// TwinCAT 3 PLC project CX9240
// ProgramVersion: 3.1.4026.20
// libraries:
//   Tc2_Standard, * (Beckhoff Automation GmbH)
//   Tc2_System, * (Beckhoff Automation GmbH)
// project tree:
//   DUTs/ ST_LED.TcDUT, ST_Switch.TcDUT, U_LED.TcDUT, U_Switch.TcDUT
//   GVLs/ GVL.TcGVL
//   / PlcTask.TcTTO
//   POUs/ MAIN.TcPOU
// real-time tasks:
//   TASK PlcTask: cycle T#10ms, priority 20, ADS port 350
//   TASK Ethernet/IP Task: cycle T#1ms, priority 2, ADS port 301
// I/O:
//   DEVICE デバイス 1 (CCAT EIP Adapter(Slave)), AmsNetId 192.168.15.13.3.1
//     Box 1 (TC EtherNet/IP Slave)
//   DEVICE デバイス 3 (EtherCAT), AmsNetId 192.168.15.13.5.1
//     ターミナル 1 (EK1200) [EK1200-5000 EtherCAT Power supply (2A E-Bus)]
//       ターミナル 3 (EL6224) [EL6224 (IO Link Master)]
//       ターミナル 4 (EK1110) [EK1110 EtherCAT extension]
//     ターミナル 5 (EK1828) [EK1828 EtherCAT IO-Coupler  (1A E-Bus, 4 Ch. Dig. In, 3ms, 8 Ch. Dig. Out 24V, 0,5A)]
//       ターミナル 6 (EL3318) [EL3318 8Ch. Ana Input Thermocouple (TC)]
//       ターミナル 6 (EL9011)
// variable links:
//   (this object) <-> Device 1 (CCAT EIP Adapter(Slave))/Box 1 (TC EtherNet/IP Slave)
//     PlcTask Inputs/GVL.uLED/uiUINT <-> Assembly 1 (Input/Output)/Inputs/uiUINT
//     PlcTask Outputs/GVL.uSwitch/uiUINT <-> Assembly 1 (Input/Output)/Outputs/uiUINT

CONFIGURATION CX9240
    RESOURCE PLC ON TwinCAT3
        TASK PlcTask(INTERVAL := T#10ms, PRIORITY := 20);
        PROGRAM MAIN WITH PlcTask : MAIN;
    END_RESOURCE
END_CONFIGURATION

// ---- DUTs/ST_LED.TcDUT
TYPE ST_LED :
STRUCT
	bGreenLED		:BIT;
	bYellowLED		:BIT;
	bRedLED			:BIT;
	bWhiteLED		:BIT;
	bBlueLED		:BIT;
END_STRUCT
END_TYPE

// ---- DUTs/ST_Switch.TcDUT
TYPE ST_Switch :
STRUCT
	bGreenSwitch		:BIT;
	bYellowSwitch		:BIT;
	bRedSwitch			:BIT;
	bWhiteSwitch		:BIT;
	bBlueSwitch			:BIT;
END_STRUCT
END_TYPE

// ---- DUTs/U_LED.TcDUT
TYPE U_LED :
UNION
	uiUINT		:UINT;
	stLED		:ST_LED;
	
END_UNION
END_TYPE

// ---- DUTs/U_Switch.TcDUT
TYPE U_Switch :
UNION
	uiUINT		:UINT;
	stSwitch	:ST_Switch;
	
END_UNION
END_TYPE

// ---- GVLs/GVL.TcGVL
{attribute 'qualified_only'}
VAR_GLOBAL
	
///---Modbus TCP---
    mb_Input_Coils					:ARRAY [0..255] OF BOOL;
    mb_Output_Coils					:ARRAY [0..255] OF BOOL;
    mb_Input_Registers				:ARRAY [0..255] OF WORD;
    mb_Output_Registers				:ARRAY [0..255] OF WORD;

//---EtherNet/IP---
	uLED					AT %I*	:U_LED;
	uSwitch					AT %Q*	:U_Switch;

END_VAR

// ---- POUs/MAIN.TcPOU
PROGRAM MAIN
VAR
END_VAR

END_PROGRAM
